{attribute 'qualified_only'}
{attribute 'strict'}
{attribute 'to_string'}
TYPE Phases :
(
	AVG 		:= 0,
	L1 			:= 1,
	L2 			:= 2,
	L3 			:= 3,
	N 			:= 4,
	minimum		:= 5,
	maximum		:= 6
) INT;
END_TYPE

(* stored: Version 1.1.0.1, ProductVersion 3.1.4024.12
   DUT Phases: Id {ed4a3401-b009-4ebd-8c5a-210cb21dcb3c} *)
